// Manual DS402 implementation
FUNCTION_BLOCK FB_MotionAxisDS402 IMPLEMENTS I_MotionAxisCommon
VAR_INPUT
END_VAR
VAR_OUTPUT
END_VAR
VAR
END_VAR

{warning 'Add property implementation'}
PROPERTY AbortDone : BOOL
GET
END_GET
END_PROPERTY

{warning 'Add property implementation'}
PROPERTY AxisState : MC_AxisStates
GET
END_GET
END_PROPERTY

{warning 'Add method implementation '}
METHOD BacklashCompensation
VAR_INPUT
    User_Enable	: BOOL;
    Backlash	: LREAL;
    BakclashRampRatio	: LREAL := 10.0;
    DisableMode	: E_DISABLEMODE := .E_DISABLEMODE.DisableModeHold;
END_VAR
END_METHOD

{warning 'Add property implementation'}
PROPERTY BufferMode : MC_BufferMode
SET
END_SET
END_PROPERTY

{warning 'Add property implementation'}
PROPERTY Busy : BOOL
GET
END_GET
END_PROPERTY

{warning 'Add property implementation'}
PROPERTY CommandAborted : BOOL
GET
END_GET
END_PROPERTY

{warning 'Add property implementation'}
PROPERTY CommandedHalt : BOOL
GET
END_GET
SET
END_SET
END_PROPERTY

{warning 'Add property implementation'}
PROPERTY CommandedMoveAbsolute : BOOL
GET
END_GET
SET
END_SET
END_PROPERTY

{warning 'Add property implementation'}
PROPERTY CommandedMoveHome : BOOL
GET
END_GET
SET
END_SET
END_PROPERTY

{warning 'Add property implementation'}
PROPERTY CommandedReset : BOOL
GET
END_GET
SET
END_SET
END_PROPERTY

{warning 'Add property implementation'}
PROPERTY EncoderCount : UDINT
GET
END_GET
END_PROPERTY

{warning 'Add property implementation'}
PROPERTY Error : BOOL
GET
END_GET
END_PROPERTY

{warning 'Add property implementation'}
PROPERTY ErrorID : UDINT
GET
END_GET
END_PROPERTY

{warning 'Add property implementation'}
PROPERTY ErrorMessage : STRING
GET
END_GET
END_PROPERTY

{warning 'Add method implementation '}
METHOD Halt
VAR_INPUT
    Execute	: BOOL;
    Deceleration	: LREAL := 0.0;
    Jerk	: LREAL := 0.0;
    BufferMode	: MC_BufferMode := .MC_BufferMode.MC_Aborting;
END_VAR
END_METHOD

{warning 'Add property implementation'}
PROPERTY HaltBufferMode : MC_BufferMode
GET
END_GET
SET
END_SET
END_PROPERTY

{warning 'Add property implementation'}
PROPERTY HaltBusy : BOOL
GET
END_GET
END_PROPERTY

{warning 'Add property implementation'}
PROPERTY HaltDeceleration : LREAL
GET
END_GET
SET
END_SET
END_PROPERTY

{warning 'Add property implementation'}
PROPERTY HaltDone : BOOL
GET
END_GET
END_PROPERTY

{warning 'Add property implementation'}
PROPERTY HaltErrorID : UDINT
GET
END_GET
END_PROPERTY

{warning 'Add property implementation'}
PROPERTY HaltJerk : LREAL
GET
END_GET
SET
END_SET
END_PROPERTY

{warning 'Add property implementation'}
PROPERTY HomeBusy : BOOL
GET
END_GET
END_PROPERTY

{warning 'Add property implementation'}
PROPERTY HomeDone : BOOL
GET
END_GET
END_PROPERTY

{warning 'Add property implementation'}
PROPERTY HomeError : BOOL
GET
END_GET
END_PROPERTY

{warning 'Add property implementation'}
PROPERTY HomeErrorID : UDINT
GET
END_GET
END_PROPERTY

{warning 'Add property implementation'}
PROPERTY HomeInterrupted : BOOL
GET
END_GET
END_PROPERTY

{warning 'Add property implementation'}
PROPERTY HomeMode : E_EpicsHomeCmd
GET
END_GET
SET
END_SET
END_PROPERTY

{warning 'Add property implementation'}
PROPERTY HomePosition : LREAL
GET
END_GET
SET
END_SET
END_PROPERTY

{warning 'Add property implementation'}
PROPERTY HomingMethod : E_DS402HomingMethod
GET
END_GET
SET
END_SET
END_PROPERTY

{warning 'Add property implementation'}
PROPERTY InTargetPosition : BOOL
GET
END_GET
END_PROPERTY

{warning 'Add property implementation'}
PROPERTY MeasuredAcceleration : LREAL
GET
END_GET
END_PROPERTY

{warning 'Add property implementation'}
PROPERTY MeasuredPosition : LREAL
GET
END_GET
END_PROPERTY

{warning 'Add property implementation'}
PROPERTY MeasuredPositionDiff : LREAL
GET
END_GET
END_PROPERTY

{warning 'Add property implementation'}
PROPERTY MeasuredVelocity : LREAL
GET
END_GET
END_PROPERTY

{warning 'Add property implementation'}
PROPERTY ModeOfOperation : SINT
GET
END_GET
SET
END_SET
END_PROPERTY

{warning 'Add method implementation '}
METHOD MoveAbsolute
VAR_INPUT
    Execute	: BOOL;
    Position	: LREAL;
    Velocity	: LREAL;
    Acceleration	: LREAL := 0.0;
    Deceleration	: LREAL := 0.0;
    Jerk	: LREAL := 0.0;
    BufferMode	: MC_BufferMode := .MC_BufferMode.MC_Aborting;
END_VAR
END_METHOD

{warning 'Add property implementation'}
PROPERTY MoveAbsoluteBusy : BOOL
GET
END_GET
END_PROPERTY

{warning 'Add property implementation'}
PROPERTY MoveAbsoluteDone : BOOL
GET
END_GET
END_PROPERTY

{warning 'Add property implementation'}
PROPERTY MoveAbsoluteError : BOOL
GET
END_GET
END_PROPERTY

{warning 'Add property implementation'}
PROPERTY MoveAbsoluteErrorID : UDINT
GET
END_GET
END_PROPERTY

{warning 'Add property implementation'}
PROPERTY MoveAbsoluteTargetAcceleration : LREAL
GET
END_GET
SET
END_SET
END_PROPERTY

{warning 'Add property implementation'}
PROPERTY MoveAbsoluteTargetDeceleration : LREAL
GET
END_GET
SET
END_SET
END_PROPERTY

{warning 'Add property implementation'}
PROPERTY MoveAbsoluteTargetJerk : LREAL
GET
END_GET
SET
END_SET
END_PROPERTY

{warning 'Add property implementation'}
PROPERTY MoveAbsoluteTargetPosition : LREAL
GET
END_GET
SET
END_SET
END_PROPERTY

{warning 'Add property implementation'}
PROPERTY MoveAbsoluteTargetVelocity : LREAL
GET
END_GET
SET
END_SET
END_PROPERTY

{warning 'Add property implementation'}
PROPERTY MoveDone : BOOL
GET
END_GET
END_PROPERTY

{warning 'Add property implementation'}
PROPERTY MoveMode : E_EpicsMotorCmd
GET
END_GET
END_PROPERTY

{warning 'Add property implementation'}
PROPERTY Name : STRING
GET
END_GET
SET
END_SET
END_PROPERTY

{warning 'Add property implementation'}
PROPERTY NCParamsReadInit : BOOL
GET
END_GET
END_PROPERTY

{warning 'Add property implementation'}
PROPERTY NegativeMotionIsEnabled : BOOL
GET
END_GET
END_PROPERTY

{warning 'Add property implementation'}
PROPERTY PositiveMotionIsEnabled : BOOL
GET
END_GET
END_PROPERTY

{warning 'Add method implementation '}
METHOD Power
VAR_INPUT
    Enable	: BOOL;
    Enable_Positive	: BOOL;
    Enable_Negative	: BOOL;
    (* in percent from 0 to 100 *)
    Override	: LREAL := 100.0;
    BufferMode	: MC_BufferMode := MC_BufferMode.MC_Aborting;
END_VAR
END_METHOD

{warning 'Add property implementation'}
PROPERTY PowerEnable : BOOL
GET
END_GET
SET
END_SET
END_PROPERTY

{warning 'Add property implementation'}
PROPERTY PowerEnableNegative : BOOL
GET
END_GET
SET
END_SET
END_PROPERTY

{warning 'Add property implementation'}
PROPERTY PowerEnablePositive : BOOL
GET
END_GET
SET
END_SET
END_PROPERTY

{warning 'Add property implementation'}
PROPERTY PowerError : BOOL
GET
END_GET
END_PROPERTY

{warning 'Add property implementation'}
PROPERTY PowerErrorID : UDINT
GET
END_GET
END_PROPERTY

{warning 'Add property implementation'}
PROPERTY PowerIsEnabled : BOOL
GET
END_GET
END_PROPERTY

{warning 'Add property implementation'}
PROPERTY PowerOverride : LREAL
GET
END_GET
SET
END_SET
END_PROPERTY

{warning 'Add property implementation'}
PROPERTY PowerStatus : BOOL
GET
END_GET
END_PROPERTY

{warning 'Add property implementation'}
PROPERTY RefreshDelay : TIME
GET
END_GET
SET
END_SET
END_PROPERTY

{warning 'Add method implementation '}
METHOD Reset
END_METHOD

{warning 'Add property implementation'}
PROPERTY ResetBusy : BOOL
GET
END_GET
END_PROPERTY

{warning 'Add property implementation'}
PROPERTY ResetDone : BOOL
GET
END_GET
END_PROPERTY

{warning 'Add property implementation'}
PROPERTY ResetError : BOOL
GET
END_GET
END_PROPERTY

{warning 'Add property implementation'}
PROPERTY ResetErrorID : UDINT
GET
END_GET
END_PROPERTY

{warning 'Add property implementation'}
PROPERTY RestoreError : BOOL
GET
END_GET
END_PROPERTY

{warning 'Add property implementation'}
PROPERTY RestoreErrorID : UDINT
GET
END_GET
END_PROPERTY

{warning 'Add property implementation'}
PROPERTY SavedPosition : LREAL
GET
END_GET
END_PROPERTY

{warning 'Add property implementation'}
PROPERTY Servo : BOOL
GET
END_GET
SET
END_SET
END_PROPERTY

{warning 'Add method implementation '}
(*
    Check all post condition before updating bCommandedMoveAbsolute
    The implmentatation will depend on the axis type
    DS402 NC/Direct axis : Implementation need to check that the drive is in the correct mode before initaiting the move then set bCommandedMoveAbsolute
    MP NC axis : will immediately write to bCommandedMoveAbsolute
*)
METHOD StartMove : BOOL
VAR_INPUT
    MoveMode	: E_EpicsMotorCmd;
    CmdExecute	: BOOL;
END_VAR
END_METHOD

END_FUNCTION_BLOCK

(* stored: Version 1.1.0.1
   POU FB_MotionAxisDS402: Id {67c0e518-0dcd-4e09-be84-2ae515d73702}, SpecialFunc None
   Property AbortDone: Id {2e545f86-a894-4584-bc4a-fe8420a5fd4a}
   Get Get: Id {7b147609-fa6c-4004-96f7-322167cf1343}
   Property AxisState: Id {8ddb7f9d-d065-48e3-ae84-bbf9768abba1}
   Get Get: Id {d8653552-9aa2-4dc7-8535-d00cf7f2be1e}
   Method BacklashCompensation: Id {2fff53ba-ccfb-4515-90fc-2151424ed910}
   Property BufferMode: Id {b04995aa-9a5d-4388-b0c3-a048d1d20653}
   Set Set: Id {e5e68606-4169-4e5a-b1ed-45968dcf5652}
   Property Busy: Id {817ec12a-fe85-4ad0-b58f-de4a61833aba}
   Get Get: Id {8b299502-0fec-4ad0-95ae-93e03f9da827}
   Property CommandAborted: Id {610c506f-0117-42ff-a26b-f404d103ce26}
   Get Get: Id {dcd4668b-2777-4ea6-adab-28ad7565d88e}
   Property CommandedHalt: Id {0c7cb23a-661b-42c8-a399-6b829d84babd}
   Get Get: Id {c92b54f6-3162-4911-bd51-6a812e092836}
   Set Set: Id {90b5bf6a-1c62-454a-a5d6-62daa11dfa65}
   Property CommandedMoveAbsolute: Id {2aeb95cc-3129-47d8-89d4-4b9aa81e5ca5}
   Get Get: Id {c5550c06-5ce0-4f65-b263-6e3501287d07}
   Set Set: Id {220937b7-0f67-4472-8b0f-e7b179b2a385}
   Property CommandedMoveHome: Id {edcf358b-9f6e-4a74-8bec-3c3f12fd5df2}
   Get Get: Id {dded372d-4a6c-4b6a-9780-dacb601491a6}
   Set Set: Id {30eac129-016e-4805-a94a-3b0f15e6b43e}
   Property CommandedReset: Id {b1242edd-d065-4924-8256-fde871362508}
   Get Get: Id {4546ccdc-803f-43e5-a29f-4c4bb9a8b845}
   Set Set: Id {bf7e82c2-c040-4297-b4a0-ae61b628ce07}
   Property EncoderCount: Id {78afa7c7-626e-4eaf-ac4c-4fcace48571f}
   Get Get: Id {bff15e72-5cce-4d46-924f-178f88e07e5f}
   Property Error: Id {7134a013-9924-4ce1-be1c-b45374707fd1}
   Get Get: Id {ab82f2a6-a175-4770-9a6a-c3f3bbc74623}
   Property ErrorID: Id {b5a03d60-8d31-4e23-ad9e-7e06637b6980}
   Get Get: Id {702858ad-944b-4c72-967c-1b5f6450942c}
   Property ErrorMessage: Id {b3ff76c4-3a00-40f8-861b-c2e93aba39e7}
   Get Get: Id {cd190f18-b024-48f0-ae7e-e615e25b3bda}
   Method Halt: Id {700ebe66-a0ff-4cec-b3ea-b56f8a615147}
   Property HaltBufferMode: Id {79ef5797-a585-4a31-8f6f-d94981bba5d1}
   Get Get: Id {168a344c-352f-4d99-8bf6-20f1b63abbf3}
   Set Set: Id {ed7582fd-4399-44df-9695-28e3b6a0da48}
   Property HaltBusy: Id {6f172334-b795-4a2a-87c8-ec742da6f167}
   Get Get: Id {2fbb836c-9a30-437d-ba54-bfd01421bcbd}
   Property HaltDeceleration: Id {e2d94a10-0340-42a5-a58b-c03dac3eca81}
   Get Get: Id {5e7e2227-f692-4f8d-a23e-125441e25a1d}
   Set Set: Id {f54c3098-f1ac-4d8a-ab29-8108e3bf50b2}
   Property HaltDone: Id {fe436c31-4a1d-4860-99f9-7eab8277ccbf}
   Get Get: Id {9c74af37-5584-4062-bee1-83d29ad29bdc}
   Property HaltErrorID: Id {f16b2591-2e85-4359-8415-91affd8d4903}
   Get Get: Id {513d7ccc-f260-4691-a6af-a7a8303171e6}
   Property HaltJerk: Id {5467fbc3-1976-4e92-a267-12043e207ae8}
   Get Get: Id {973a2718-2c37-4b2d-966d-ec42746e9818}
   Set Set: Id {835f658a-550e-43bd-83f3-e1f134ef4816}
   Property HomeBusy: Id {f323546b-d4dc-4e60-bf27-aceeed771c24}
   Get Get: Id {23777cd3-163f-459b-acca-36c33dbedba2}
   Property HomeDone: Id {86b1387b-d004-4d2c-9bfe-d21e043d7e03}
   Get Get: Id {d1efa01c-d984-40c1-b113-7de71f343c3d}
   Property HomeError: Id {8702416c-80f1-4239-8c2c-a47851dc8921}
   Get Get: Id {c3010afd-8e0f-4e58-b2e4-bb200da34c13}
   Property HomeErrorID: Id {c18c3bd8-0453-49da-9e73-2a992c86e6b7}
   Get Get: Id {86f7c806-48c3-40f0-b561-bbc3d9aeeb62}
   Property HomeInterrupted: Id {f31951bd-3235-4b77-beeb-0519587a5c80}
   Get Get: Id {eb3cbe17-ce67-494c-9103-f7b83a99f1b2}
   Property HomeMode: Id {14c1c98d-a0e2-42b3-87eb-47fd58fabe10}
   Get Get: Id {04e5056b-9b36-433d-b6af-d57d18be1329}
   Set Set: Id {68e1bcaa-8f6d-491f-a970-fbdf6a31d9e2}
   Property HomePosition: Id {41785016-7d21-41b4-a540-a63933d0f65a}
   Get Get: Id {85a30268-471d-4d7d-8247-aba7b443ce1e}
   Set Set: Id {28b4d882-2bde-489e-8a77-ae3bcf3c41ed}
   Property HomingMethod: Id {f2289d60-652e-44f7-8e57-651a4c02a4f6}
   Get Get: Id {047bc289-3d68-4aee-a2e5-ead5fd43a87d}
   Set Set: Id {ca2af230-19eb-4da2-9943-91c2012102d1}
   Property InTargetPosition: Id {78bcbc79-ed88-441a-a19a-d3d0af8a3a81}
   Get Get: Id {ba6a7530-eb38-4bcd-a985-b0485691111e}
   Property MeasuredAcceleration: Id {c44ed0e9-967e-4602-93ed-f14054a337b9}
   Get Get: Id {b6b7364a-f788-4c78-85e1-523ecc47cfb7}
   Property MeasuredPosition: Id {7fad4265-be4a-4969-8d3e-0546c649470f}
   Get Get: Id {f67204fc-dcdb-4ef8-9c7f-94f35d568e2a}
   Property MeasuredPositionDiff: Id {17950501-03c9-4e16-ab2d-c6160ea00862}
   Get Get: Id {a2f4267a-b15c-45c7-8dec-e7d636a926f3}
   Property MeasuredVelocity: Id {ff5da3c8-0e27-422a-abde-e1ea759a0be5}
   Get Get: Id {56050aa3-7a73-432d-bef7-874b1782065c}
   Property ModeOfOperation: Id {49445804-602f-40f7-b896-4ef26d6c2703}
   Get Get: Id {64e75829-32e7-4f37-9b36-75dfc3974c33}
   Set Set: Id {a8ef1067-f6df-4cb5-8f8f-0dad5309bcb8}
   Method MoveAbsolute: Id {bba99ede-4b2c-4fa9-8d0d-e57085d22ce7}
   Property MoveAbsoluteBusy: Id {d5977205-b583-4298-86c8-52abba69e9a3}
   Get Get: Id {25740a77-f258-4f83-86c6-817992c57ff9}
   Property MoveAbsoluteDone: Id {4ba4b3cd-bef0-437b-aad1-eea291cdc568}
   Get Get: Id {40aeb904-a7cd-4a25-9b57-fcc0a225e202}
   Property MoveAbsoluteError: Id {d917724a-8181-42fb-bd2a-8fa7b157100d}
   Get Get: Id {a543248b-5376-4b43-8257-10d027bf19fc}
   Property MoveAbsoluteErrorID: Id {6a8a05f7-afe0-4712-baff-be2090ea98f4}
   Get Get: Id {891d1fcb-3717-4c9b-a3b3-e5216d6fb799}
   Property MoveAbsoluteTargetAcceleration: Id {43116dca-55a8-454f-a3ad-85b9ad4c8d9a}
   Get Get: Id {ac461724-fda1-4d8b-ac05-3e173964bf91}
   Set Set: Id {27a00e86-c295-44f4-9564-98fe093ff27a}
   Property MoveAbsoluteTargetDeceleration: Id {64058680-3497-46c6-9271-2d2540a0c23d}
   Get Get: Id {9ca66405-95d6-413f-875a-f282b4aa0130}
   Set Set: Id {e10fa46f-0157-4cb6-bb31-717b0c5894ce}
   Property MoveAbsoluteTargetJerk: Id {dbeb6034-c325-4385-8649-85a0156ff85c}
   Get Get: Id {2062e8be-a10c-4ccb-9255-f847097ddc91}
   Set Set: Id {1ad2a428-e28a-4225-b2a9-8e971ed601e9}
   Property MoveAbsoluteTargetPosition: Id {691413be-d0f9-4441-a343-97e1508bcd0d}
   Get Get: Id {c1344c95-faad-48c9-bd7a-7a2abd0eb777}
   Set Set: Id {83f01970-3f8e-4e13-8598-a8bbee54076e}
   Property MoveAbsoluteTargetVelocity: Id {34c5ef46-22f8-40bf-bf44-4f3746739228}
   Get Get: Id {f9cb781d-fa3e-4e71-b484-cedcc416e797}
   Set Set: Id {e391282b-cd45-4704-84cd-e82b8633ecf1}
   Property MoveDone: Id {4dc97363-5124-4f5e-8161-9b629560161c}
   Get Get: Id {fb3b96a6-5e09-4d1c-a936-83126497aa3a}
   Property MoveMode: Id {e243a820-eda8-4928-936c-381abbdaf3a3}
   Get Get: Id {d3717b38-8e53-4c0d-90d4-89d110d6b399}
   Property Name: Id {b6cb0e39-3a14-4bde-9bd5-b8a8340e19dd}
   Get Get: Id {120e1a29-635c-474e-b9ab-344834feeda6}
   Set Set: Id {1612b255-bfce-4b4f-870d-5c10ca36db98}
   Property NCParamsReadInit: Id {b13880cf-a9ae-4a36-9506-c2c43a523116}
   Get Get: Id {b84cbc31-0bb8-4d89-b77b-e129c0dd716c}
   Property NegativeMotionIsEnabled: Id {e48d0963-f75b-4bad-90f3-fcfbcf4dabcd}
   Get Get: Id {0778e913-15d2-4a6f-af82-4329e6194164}
   Property PositiveMotionIsEnabled: Id {ff377bbb-2d82-4db4-b4d6-73dbfe4f874c}
   Get Get: Id {825be891-e6e3-41dc-ab85-47267b266a2b}
   Method Power: Id {58da6095-9f7d-4c3a-9f07-2e2e032ac15f}
   Property PowerEnable: Id {eed9482d-9b64-44f4-857f-0e08ca0fa04f}
   Get Get: Id {4c4b372f-2864-46f0-a9ea-525b014daa6a}
   Set Set: Id {a069b200-b6ef-4530-b2f9-1dd914551559}
   Property PowerEnableNegative: Id {a24b0d20-be2e-4eba-b9b2-51e833f992d1}
   Get Get: Id {e8a52dfc-b6b2-4c40-87da-587494509b03}
   Set Set: Id {0c71330e-a60a-4582-ac0d-d2dc5757f11f}
   Property PowerEnablePositive: Id {68fd1536-5e35-4e77-9d69-3cd4989bdbc3}
   Get Get: Id {5f67944d-fca2-49a2-b42a-682949502873}
   Set Set: Id {e63529ae-c5e6-4e7d-8f1c-d9d8ca1eb7c9}
   Property PowerError: Id {ecd9a068-5caf-4701-bebe-c01834045247}
   Get Get: Id {88ecba80-bff5-4af8-855f-3d377ccaa9c1}
   Property PowerErrorID: Id {35f75f88-4cb2-4f44-babd-aa3f4cdeacb4}
   Get Get: Id {dc4d263c-2c89-4b20-885a-909cfadbf2b2}
   Property PowerIsEnabled: Id {1146c417-4136-42c0-8ad9-56e7b7e54639}
   Get Get: Id {12e15921-1d58-468a-b1dd-b2da18419dd2}
   Property PowerOverride: Id {ff06008b-6c10-49ad-8fad-e6f511e88c80}
   Get Get: Id {a5ef008e-9bc7-431f-ae7f-b6e1c594b65b}
   Set Set: Id {e596b239-24fa-4b8a-a66e-15d1693e0b68}
   Property PowerStatus: Id {43056afd-589f-4d8f-abf8-0aa6e320a894}
   Get Get: Id {ae599094-1201-4fd5-b1ab-cc39ff1c794e}
   Property RefreshDelay: Id {2990b3e3-5295-4e77-bc18-ca861e49db15}
   Get Get: Id {0d57a54f-d422-4918-8090-3d52682a728e}
   Set Set: Id {f700d883-a9fa-4a2d-a27c-5a1e919b9dbb}
   Method Reset: Id {b8fb4790-72b4-4cab-a1b4-c5420e6448bc}
   Property ResetBusy: Id {e2236231-6bde-4856-a0be-a9d4e2753eef}
   Get Get: Id {4307ce23-8e20-4251-b3cf-d4ef359658a0}
   Property ResetDone: Id {41ffa7f7-20ec-4134-ac87-5390f76484a3}
   Get Get: Id {a9b34ee8-56c5-4493-94cb-d346f06fc16b}
   Property ResetError: Id {33040d73-646c-4c68-8b4c-cd05b8eb8ef6}
   Get Get: Id {88197e08-f10c-41f5-8b34-81cdd87e4ec6}
   Property ResetErrorID: Id {f30da60b-da33-4e44-b5ec-9de92cb70d7e}
   Get Get: Id {694c11fd-1398-4678-bd5c-3c7426ee3337}
   Property RestoreError: Id {70fa072e-2ec9-4e05-8e47-4be6413da6ac}
   Get Get: Id {c97c6671-7f07-4d52-99c1-f8c1de9e1a42}
   Property RestoreErrorID: Id {bd37587e-f283-4fd4-a477-2f5ab3c69656}
   Get Get: Id {7041f7d7-1692-4b75-b356-ca9c6dda63cb}
   Property SavedPosition: Id {72e41ee6-9b2a-4be3-8da6-cabb839ab689}
   Get Get: Id {3925a432-8e1d-402b-9606-25024effe5f7}
   Property Servo: Id {eed722ea-cc3c-41d1-85e7-1a696d153f62}
   Get Get: Id {4894b852-6ae6-48a1-97ba-2060451a64d0}
   Set Set: Id {92ac422a-4db0-430c-9867-0cdf5ce1ca35}
   Method StartMove: Id {d71a5e48-7e3e-476d-937f-032541c0cb1a} *)
